{attribute 'qualified_only'}
{attribute 'strict'}
{attribute 'to_string'}
TYPE ARCommunicationValueType_t :
(
	NUMBER := 0,
	TEXT,
	BOOLEAN
);
END_TYPE

(* stored: Version 1.1.0.1
   DUT ARCommunicationValueType_t: Id {cb1d9388-322d-4a94-9d4d-c8c7b30cdbb6} *)
